FUNCTION_BLOCK Basic1 (* Basic Function Block Type *)
  (* Standard: 61499-2 *)
  (* Version 0.0, 24/05/2016, Chen-Wei, nxtControl GmbH, Template *)
  PACKAGE Main;
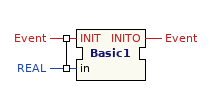
  EVENT_INPUT
    INIT WITH in; (* Initialization Request *)
  END_EVENT
  EVENT_OUTPUT
    INITO; (* Initialization Confirm *)
  END_EVENT
  VAR_INPUT
    in : REAL;
  END_VAR
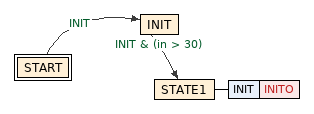
  EC_STATES
    START; (* Initial State *)
    INIT; (* Initialization *)
    STATE1 : INIT -> INITO;
  END_STATES
  EC_TRANSITIONS
    START TO INIT := INIT;
    INIT TO STATE1 := INIT & (in > 30);
  END_TRANSITIONS
  ALGORITHM INIT IN ST: (* Initialization algorithm *)
;
  END_ALGORITHM
  ALGORITHM REQ IN ST: (* Normally executed algorithm *)
;
  END_ALGORITHM
END_FUNCTION_BLOCK
